FUNCTION_BLOCK SS3_ps_Camera (* Composite FB wrapping other FBs *)
  (* Standard: 61499-2 *)
  (* Version 1.0, 2025-08-24, PS_Transformer_for_Unknown *)
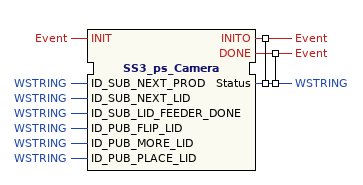
  EVENT_INPUT
    INIT; (* Initialization Request *)
  END_EVENT
  EVENT_OUTPUT
    INITO WITH Status; (* Initialization Confirm *)
    DONE WITH Status; (* Execution Confirmation *)
  END_EVENT
  VAR_INPUT
    ID_SUB_NEXT_PROD : WSTRING;
    ID_SUB_NEXT_LID : WSTRING;
    ID_SUB_LID_FEEDER_DONE : WSTRING;
    ID_PUB_FLIP_LID : WSTRING;
    ID_PUB_MORE_LID : WSTRING;
    ID_PUB_PLACE_LID : WSTRING;
  END_VAR
  VAR_OUTPUT
    Status : WSTRING; (* Output event qualifier *)
  END_VAR
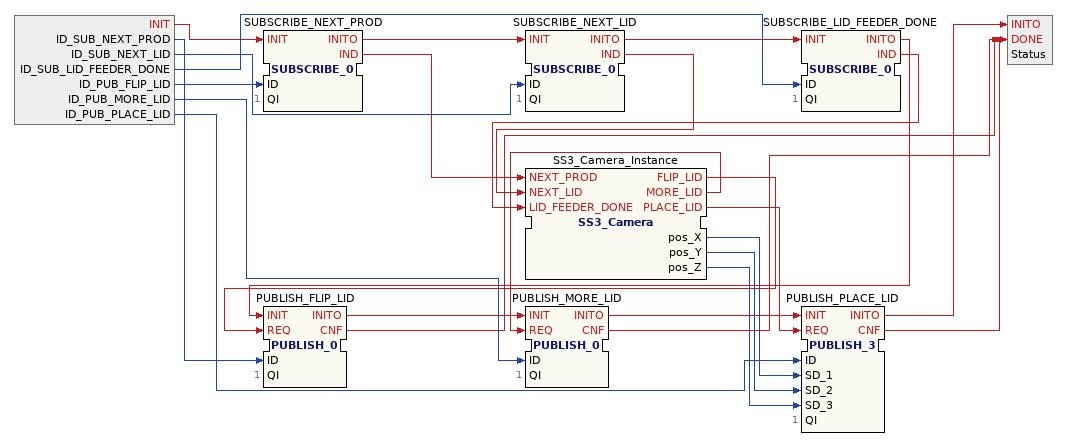
  FBS
    SS3_Camera_Instance : SS3_Camera;
    SUBSCRIBE_NEXT_PROD : SUBSCRIBE_0(QI := 1);
    SUBSCRIBE_NEXT_LID : SUBSCRIBE_0(QI := 1);
    SUBSCRIBE_LID_FEEDER_DONE : SUBSCRIBE_0(QI := 1);
    PUBLISH_FLIP_LID : PUBLISH_0(QI := 1);
    PUBLISH_MORE_LID : PUBLISH_0(QI := 1);
    PUBLISH_PLACE_LID : PUBLISH_3(QI := 1);
  END_FBS
  EVENT_CONNECTIONS
    INIT TO SUBSCRIBE_NEXT_PROD.INIT;
    SUBSCRIBE_NEXT_PROD.INITO TO SUBSCRIBE_NEXT_LID.INIT;
    SUBSCRIBE_NEXT_LID.INITO TO SUBSCRIBE_LID_FEEDER_DONE.INIT;
    SUBSCRIBE_LID_FEEDER_DONE.INITO TO PUBLISH_FLIP_LID.INIT;
    PUBLISH_FLIP_LID.INITO TO PUBLISH_MORE_LID.INIT;
    PUBLISH_MORE_LID.INITO TO PUBLISH_PLACE_LID.INIT;
    PUBLISH_PLACE_LID.INITO TO INITO;
    SUBSCRIBE_NEXT_PROD.IND TO SS3_Camera_Instance.NEXT_PROD;
    SUBSCRIBE_NEXT_LID.IND TO SS3_Camera_Instance.NEXT_LID;
    SUBSCRIBE_LID_FEEDER_DONE.IND TO SS3_Camera_Instance.LID_FEEDER_DONE;
    SS3_Camera_Instance.FLIP_LID TO PUBLISH_FLIP_LID.REQ;
    SS3_Camera_Instance.MORE_LID TO PUBLISH_MORE_LID.REQ;
    SS3_Camera_Instance.PLACE_LID TO PUBLISH_PLACE_LID.REQ;
    PUBLISH_FLIP_LID.CNF TO DONE;
    PUBLISH_MORE_LID.CNF TO DONE;
    PUBLISH_PLACE_LID.CNF TO DONE;
  END_CONNECTIONS
  DATA_CONNECTIONS
    ID_SUB_NEXT_PROD TO SUBSCRIBE_NEXT_PROD.ID;
    ID_SUB_NEXT_LID TO SUBSCRIBE_NEXT_LID.ID;
    ID_SUB_LID_FEEDER_DONE TO SUBSCRIBE_LID_FEEDER_DONE.ID;
    ID_PUB_FLIP_LID TO PUBLISH_FLIP_LID.ID;
    ID_PUB_MORE_LID TO PUBLISH_MORE_LID.ID;
    ID_PUB_PLACE_LID TO PUBLISH_PLACE_LID.ID;
    SS3_Camera_Instance.pos_X TO PUBLISH_PLACE_LID.SD_1;
    SS3_Camera_Instance.pos_Y TO PUBLISH_PLACE_LID.SD_2;
    SS3_Camera_Instance.pos_Z TO PUBLISH_PLACE_LID.SD_3;
  END_CONNECTIONS
END_FUNCTION_BLOCK
